// Mitsubishi GX Works2 project: IHW4   PLC: Q03UDE

// global labels: Global1
VAR_GLOBAL
  STARTBUTTON AT X40 : BOOL;
  STOPBUTTON AT X41 : BOOL;
  ESTOPBUTTON AT X42 : BOOL;
  DTRUONG AT Y50 : BOOL;
  DDAI AT Y51 : BOOL;
  DHOC AT Y52 : BOOL;
  DCONG AT Y53 : BOOL;
  DNGHIEP AT Y54 : BOOL;
  DHA AT Y55 : BOOL;
  DNOI AT Y56 : BOOL;
END_VAR

PROGRAM MAIN
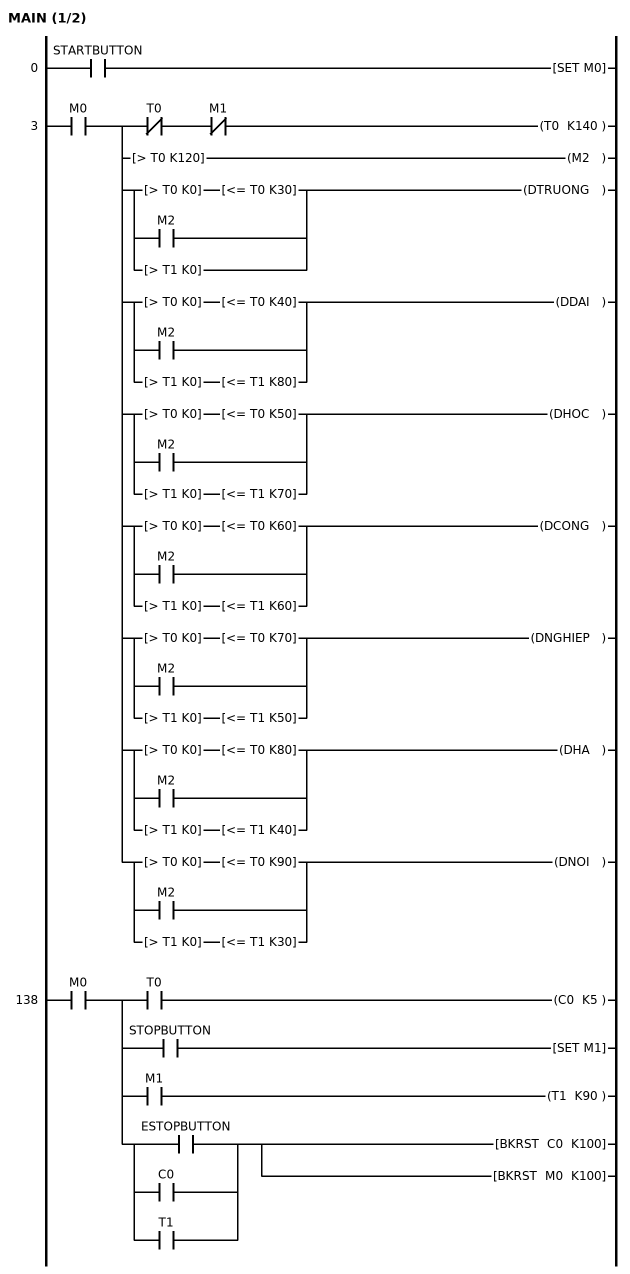
0     LD      STARTBUTTON
      SET     M0
3     LD      M0
      MPS
      ANI     T0
      ANI     M1
      OUT     T0 K140
      MRD
      AND>    T0 K120
      OUT     M2
      MRD
      LD>     T0 K0
      AND<=   T0 K30
      OR      M2
      OR>     T1 K0
      ANB
      OUT     DTRUONG
      MRD
      LD>     T0 K0
      AND<=   T0 K40
      OR      M2
      LD>     T1 K0
      AND<=   T1 K80
      ORB
      ANB
      OUT     DDAI
      MRD
      LD>     T0 K0
      AND<=   T0 K50
      OR      M2
      LD>     T1 K0
      AND<=   T1 K70
      ORB
      ANB
      OUT     DHOC
      MRD
      LD>     T0 K0
      AND<=   T0 K60
      OR      M2
      LD>     T1 K0
      AND<=   T1 K60
      ORB
      ANB
      OUT     DCONG
      MRD
      LD>     T0 K0
      AND<=   T0 K70
      OR      M2
      LD>     T1 K0
      AND<=   T1 K50
      ORB
      ANB
      OUT     DNGHIEP
      MRD
      LD>     T0 K0
      AND<=   T0 K80
      OR      M2
      LD>     T1 K0
      AND<=   T1 K40
      ORB
      ANB
      OUT     DHA
      MPP
      LD>     T0 K0
      AND<=   T0 K90
      OR      M2
      LD>     T1 K0
      AND<=   T1 K30
      ORB
      ANB
      OUT     DNOI
138   LD      M0
      MPS
      AND     T0
      OUT     C0 K5
      MRD
      AND     STOPBUTTON
      SET     M1
      MRD
      AND     M1
      OUT     T1 K90
      MPP
      LD      ESTOPBUTTON
      OR      C0
      OR      T1
      ANB
      BKRST   C0 K100
      BKRST   M0 K100
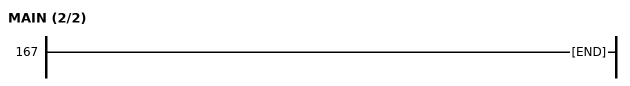
167   END
END_PROGRAM
